{attribute 'pack_mode' := '2'}
TYPE U_STATION_CTRL :
UNION  
  _st           : ARRAY[1..MAX_STATION] OF ST_STATION_CTRL;
  _by   AT %Q*  : ARRAY[1..MAX_STATION] OF
                  ARRAY[1..SIZEOF(ST_STATION_CTRL)] OF BYTE;
END_UNION
END_TYPE

(* stored: Version 1.1.0.1, ProductVersion 3.1.4024.12
   DUT U_STATION_CTRL: Id {737ed184-4012-4cb6-897f-3a5d68c7357f} *)
